FUNCTION "LGF_StringToInt" : DInt
TITLE = LGF_StringToInt
{ S7_Optimized_Access := 'TRUE' }
AUTHOR : Siemens_Digital_Industry
FAMILY : LGF
NAME : LGF_StringToInt
//This function converts a variable of data type `String` into a variable of data type `DInt`.
   VAR_INPUT
      value : String;   // String value to be converted to Double-Integer.  Example: ‘+16927’
   END_VAR

   VAR_TEMP
      tempDoubleInteger : DInt;   // Temp DInt value for conversion from String
   END_VAR

   VAR CONSTANT
      CONVERT_FORMAT_TO_INTEGER : Word := 16#0000;   // Input format of the characters - Decimal fraction "."
      CONVERT_START_POSITION : UInt := 1;   // Reference to the first character to be converted - first character = 1
   END_VAR


BEGIN
	REGION BLOCK INFO HEADER
	  //===============================================================================
	  // SIEMENS AG / (c)Copyright 2019
	  //-------------------------------------------------------------------------------
	  // Title:            LGF_StringToInt
	  // Comment/Function: This function converts a string to an integer value
	  //                   Vice versa of the LGF_IntToString - wrapper of the system function VAL_STRG.
	  // Library/Family:   LGF(Library General Functions)
	  // Author:           Siemens Digital Industry Support
	  // Tested with:
	  // Engineering:      TIA Portal V15.1
	  // Restrictions:     ENO handling done by STRG_VAL
	  // Requirements:     PLC (S7-1200 / S7-1500)
	  //-------------------------------------------------------------------------------
	  // Change log table:
	  // Version  | Date       | Expert in charge       | Changes applied
	  //----------|------------|------------------------|------------------------------
	  // 01.00.01 | 12.06.2019 | Simatic Systems Support
	  //                         First released version
	  // 01.00.03 | 30.07.2019 | Simatic Systems Support
	  //                         Add ENO handling
	  // 03.00.00 | 23.04.2020 | Simatic Systems Support | Set version to V3.0.0
	  //                         Harmonize the version of the whole library
	  // 03.00.01 | 23.02.2021 | Simatic Systems Support
	  //                         Insert documentation
	  //                         ENO handling done by STRG_VAL system function
	  //===============================================================================
	END_REGION Block info header

	REGION CONVERSION
	  STRG_VAL(IN     := #value,
	           FORMAT := #CONVERT_FORMAT_TO_INTEGER,
	           P      := #CONVERT_START_POSITION,
	           OUT    => #tempDoubleInteger);
	END_REGION

	REGION OUTPUT
	  #LGF_StringToInt := #tempDoubleInteger;
	END_REGION

END_FUNCTION

